// Mitsubishi GX Works2 project: Ladder estruturado   PLC: Q03UDV

// task Task_01 (event TRUE, interval 0, priority 31): POU_01

PROGRAM POU_01
VAR
  CTD_1 : CTD;
  CTU_1 : CTU;
  CTUD_1 : CTUD;
  TP_1 : TP;
  TON_1 : TON;
  TOF_1 : TOF;
  TimeTP : TIME;
  TimeON : TIME;
  TimeOFF : TIME;
  TP_2 : TP;
END_VAR
(* structured ladder/FBD written out as ST: instructions are called as NAME(EN, inputs, outputs); _pN, _eN, _tN stand for wires *)
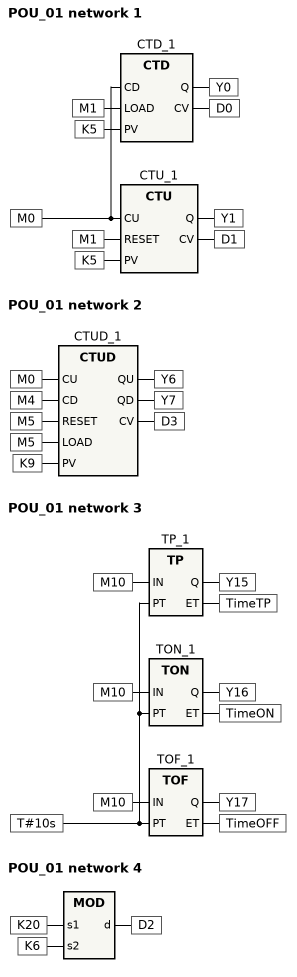
(* network 1 *)
CTD_1(CD := M0, LOAD := M1, PV := K5, Q => Y0, CV => D0);
CTU_1(CU := M0, RESET := M1, PV := K5, Q => Y1, CV => D1);
(* network 2 *)
CTUD_1(CU := M0, CD := M4, RESET := M5, LOAD := M5, PV := K9, QU => Y6, QD => Y7, CV => D3);
(* network 3 *)
TP_1(IN := M10, PT := T#10s, Q => Y15, ET => TimeTP);
TON_1(IN := M10, PT := T#10s, Q => Y16, ET => TimeON);
TOF_1(IN := M10, PT := T#10s, Q => Y17, ET => TimeOFF);
(* network 4 *)
D2 := MOD(K20, K6);
END_PROGRAM
